// TwinCAT 3 PLC project CoreExample
// ProgramVersion: 3.1.4026.17
// libraries:
//   Tc2_Standard, * (Beckhoff Automation GmbH)
//   Tc2_System, * (Beckhoff Automation GmbH)
//   Tc3_JsonXml, * (Beckhoff Automation GmbH)
//   Tc3_Module, * (Beckhoff Automation GmbH)
//   [Twincat Open Library], * (Home)
//   VisuSymbols,3.5.10.0,System
// project tree:
//   DUTs/ ST_CameraStates.TcDUT (not stored)
//   GVLs/ Hardware_Mapping.TcGVL (not stored), Cognex_Mapping.TcGVL (not stored)
//   / PlcTask.TcTTO (not stored)
//   POUs/ MAIN.TcPOU, _5000_PRG_Aborting.TcPOU, _1000_PRG_Homing.TcPOU, _3000_PRG_Running.TcPOU, _2000_PRG_Stopping.TcPOU, _4000_PRG_Pausing.TcPOU, _6000_PRG_Proceeding.TcPOU
// real-time tasks:
//   TASK PlcTask: cycle T#10ms, priority 20, ADS port 350
//   TASK VISU_TASK: cycle T#200000us, priority 30, ADS port 351
//   TASK IO Task New: cycle T#1ms, priority 1, ADS port 301
// motion (NC):
//   TASK NC-Task 1 SAF: cycle T#2ms, priority 4, ADS port 501
//   TASK NC-Task 1 SVB: cycle T#10ms, priority 8, ADS port 511
//   AXIS Axis 1 (id 1)
//     OtherSettings: AllowMotionCmdToSlave=true
//     encoder EncType=4
//       EncPara: MaxCount=#x0000ffff
//         Inc: RefSoftSyncMask=#x0000ffff
//     drive DrvType=24
//       Analog: TorqueSetpointScale=10, ScaleFactorActTorque=0.1
//       TimeComp: TaskDelayCycles=1
//     controller CtrType=1
//       CtrPara: PriorControlFactor=1
//         Observer: BandWidth=20
//   AXIS Axis 2 (id 2)
//     OtherSettings: AllowMotionCmdToSlave=true
//     encoder EncType=4
//       EncPara: MaxCount=#x0000ffff
//         Inc: RefSoftSyncMask=#x0000ffff
//     drive DrvType=24
//       Analog: TorqueSetpointScale=10, ScaleFactorActTorque=0.1
//       TimeComp: TaskDelayCycles=1
//     controller CtrType=1
//       CtrPara: PriorControlFactor=1
//         Observer: BandWidth=20
// I/O:
//   DEVICE Device 1 (TC3 EIP Scanner), AmsNetId 172.18.236.100.2.1
//     Box 1 (In-Sight 7000 Series) // <INFO> </INFO> <EDS> C:\TwinCAT\3.1\Config\Io\EtherNetIP\02A6006401090C00.eds </EDS>
//   DEVICE Device 2 (EtherCAT), AmsNetId 172.18.236.100.3.1
//     Term 2 (EK1100) [EK1100 EtherCAT Coupler (2A E-Bus)]
//       Term 3 (EL1008) [EL1008 8Ch. Dig. Input 24V, 3ms]
//       Term 4 (EL1008) [EL1008 8Ch. Dig. Input 24V, 3ms]
//       Term 5 (EL2008) [EL2008 8Ch. Dig. Output 24V, 0.5A]
//       Term 6 (EL2008) [EL2008 8Ch. Dig. Output 24V, 0.5A]
//       Term 7 (EL7047) [EL7047 1Ch. Stepper motor output stage (50V, 5A)]
//       Term 8 (EL7047) [EL7047 1Ch. Stepper motor output stage (50V, 5A)]
//       Term 8 (EL9011) [EL9011 End Terminal]
// variable links:
//   NC-Task 1 SAF/Axes/Axis 1 <-> Device 2 (EtherCAT)/Term 2 (EK1100)/Term 7 (EL7047)
//     Drive/Inputs/In/nState1 @bit 3 <-> STM Status/Status/Error
//     Drive/Inputs/In/nState1 @bit 7 <-> STM Status/Status/Motor stall
//     Drive/Inputs/In/nState1 @bit 5 <-> STM Status/Status/Moving negative
//     Drive/Inputs/In/nState1 @bit 4 <-> STM Status/Status/Moving positive
//     Drive/Inputs/In/nState1 @bit 1 <-> STM Status/Status/Ready
//     Drive/Inputs/In/nState1 <-> STM Status/Status/Ready to enable
//     Drive/Inputs/In/nState1 @bit 6 <-> STM Status/Status/Torque reduced
//     Drive/Inputs/In/nState1 @bit 2 <-> STM Status/Status/Warning
//     Drive/Inputs/In/nState2 @bit 3 <-> STM Status/Status/Digital input 1
//     Drive/Inputs/In/nState2 @bit 4 <-> STM Status/Status/Digital input 2
//     Drive/Inputs/In/nState2 @bit 5 <-> STM Status/Status/Sync error
//     Drive/Inputs/In/nState2 @bit 7 <-> STM Status/Status/TxPDO Toggle
//     Drive/Inputs/In/nState4 @bit 1 <-> WcState/InputToggle
//     Drive/Inputs/In/nState4 <-> WcState/WcState
//     Drive/Outputs/Out/nCtrl1 <-> STM Control/Control/Enable
//     Drive/Outputs/Out/nCtrl1 @bit 2 <-> STM Control/Control/Reduce torque
//     Drive/Outputs/Out/nCtrl1 @bit 1 <-> STM Control/Control/Reset
//     Drive/Outputs/Out/nCtrl2 @bit 3 <-> STM Control/Control/Digital output 1
//     Drive/Outputs/Out/nDataOut2[0] <-> STM Velocity/Velocity
//     Enc/Inputs/In/nDataIn1[0] <-> ENC Status compact/Counter value
//     Enc/Inputs/In/nDataIn2[0] <-> ENC Status compact/Latch value
//     Enc/Inputs/In/nState1 @bit 4 <-> ENC Status compact/Status/Counter overflow
//     Enc/Inputs/In/nState1 @bit 3 <-> ENC Status compact/Status/Counter underflow
//     Enc/Inputs/In/nState1 @bit 7 <-> ENC Status compact/Status/Extrapolation stall
//     Enc/Inputs/In/nState1 <-> ENC Status compact/Status/Latch C valid
//     Enc/Inputs/In/nState1 @bit 1 <-> ENC Status compact/Status/Latch extern valid
//     Enc/Inputs/In/nState1 @bit 2 <-> ENC Status compact/Status/Set counter done
//     Enc/Inputs/In/nState2 @bit 4 <-> ENC Status compact/Status/Status of extern latch
//     Enc/Inputs/In/nState2 <-> ENC Status compact/Status/Status of input A
//     Enc/Inputs/In/nState2 @bit 1 <-> ENC Status compact/Status/Status of input B
//     Enc/Inputs/In/nState2 @bit 2 <-> ENC Status compact/Status/Status of input C
//     Enc/Inputs/In/nState2 @bit 5 <-> ENC Status compact/Status/Sync error
//     Enc/Inputs/In/nState2 @bit 7 <-> ENC Status compact/Status/TxPDO Toggle
//     Enc/Inputs/In/nState4 @bit 1 <-> WcState/InputToggle
//     Enc/Inputs/In/nState4 <-> WcState/WcState
//     Enc/Outputs/Out/nCtrl1 <-> ENC Control compact/Control/Enable latch C
//     Enc/Outputs/Out/nCtrl1 @bit 3 <-> ENC Control compact/Control/Enable latch extern on negative edge
//     Enc/Outputs/Out/nCtrl1 @bit 1 <-> ENC Control compact/Control/Enable latch extern on positive edge
//     Enc/Outputs/Out/nCtrl1 @bit 2 <-> ENC Control compact/Control/Set counter
//     Enc/Outputs/Out/nDataOut1[0] <-> ENC Control compact/Set counter value
//   NC-Task 1 SAF/Axes/Axis 2 <-> Device 2 (EtherCAT)/Term 2 (EK1100)/Term 8 (EL7047)
//     Drive/Inputs/In/nState1 @bit 3 <-> STM Status/Status/Error
//     Drive/Inputs/In/nState1 @bit 7 <-> STM Status/Status/Motor stall
//     Drive/Inputs/In/nState1 @bit 5 <-> STM Status/Status/Moving negative
//     Drive/Inputs/In/nState1 @bit 4 <-> STM Status/Status/Moving positive
//     Drive/Inputs/In/nState1 @bit 1 <-> STM Status/Status/Ready
//     Drive/Inputs/In/nState1 <-> STM Status/Status/Ready to enable
//     Drive/Inputs/In/nState1 @bit 6 <-> STM Status/Status/Torque reduced
//     Drive/Inputs/In/nState1 @bit 2 <-> STM Status/Status/Warning
//     Drive/Inputs/In/nState2 @bit 3 <-> STM Status/Status/Digital input 1
//     Drive/Inputs/In/nState2 @bit 4 <-> STM Status/Status/Digital input 2
//     Drive/Inputs/In/nState2 @bit 5 <-> STM Status/Status/Sync error
//     Drive/Inputs/In/nState2 @bit 7 <-> STM Status/Status/TxPDO Toggle
//     Drive/Inputs/In/nState4 @bit 1 <-> WcState/InputToggle
//     Drive/Inputs/In/nState4 <-> WcState/WcState
//     Drive/Outputs/Out/nCtrl1 <-> STM Control/Control/Enable
//     Drive/Outputs/Out/nCtrl1 @bit 2 <-> STM Control/Control/Reduce torque
//     Drive/Outputs/Out/nCtrl1 @bit 1 <-> STM Control/Control/Reset
//     Drive/Outputs/Out/nCtrl2 @bit 3 <-> STM Control/Control/Digital output 1
//     Drive/Outputs/Out/nDataOut2[0] <-> STM Velocity/Velocity
//     Enc/Inputs/In/nDataIn1[0] <-> ENC Status compact/Counter value
//     Enc/Inputs/In/nDataIn2[0] <-> ENC Status compact/Latch value
//     Enc/Inputs/In/nState1 @bit 4 <-> ENC Status compact/Status/Counter overflow
//     Enc/Inputs/In/nState1 @bit 3 <-> ENC Status compact/Status/Counter underflow
//     Enc/Inputs/In/nState1 @bit 7 <-> ENC Status compact/Status/Extrapolation stall
//     Enc/Inputs/In/nState1 <-> ENC Status compact/Status/Latch C valid
//     Enc/Inputs/In/nState1 @bit 1 <-> ENC Status compact/Status/Latch extern valid
//     Enc/Inputs/In/nState1 @bit 2 <-> ENC Status compact/Status/Set counter done
//     Enc/Inputs/In/nState2 @bit 4 <-> ENC Status compact/Status/Status of extern latch
//     Enc/Inputs/In/nState2 <-> ENC Status compact/Status/Status of input A
//     Enc/Inputs/In/nState2 @bit 1 <-> ENC Status compact/Status/Status of input B
//     Enc/Inputs/In/nState2 @bit 2 <-> ENC Status compact/Status/Status of input C
//     Enc/Inputs/In/nState2 @bit 5 <-> ENC Status compact/Status/Sync error
//     Enc/Inputs/In/nState2 @bit 7 <-> ENC Status compact/Status/TxPDO Toggle
//     Enc/Inputs/In/nState4 @bit 1 <-> WcState/InputToggle
//     Enc/Inputs/In/nState4 <-> WcState/WcState
//     Enc/Outputs/Out/nCtrl1 <-> ENC Control compact/Control/Enable latch C
//     Enc/Outputs/Out/nCtrl1 @bit 3 <-> ENC Control compact/Control/Enable latch extern on negative edge
//     Enc/Outputs/Out/nCtrl1 @bit 1 <-> ENC Control compact/Control/Enable latch extern on positive edge
//     Enc/Outputs/Out/nCtrl1 @bit 2 <-> ENC Control compact/Control/Set counter
//     Enc/Outputs/Out/nDataOut1[0] <-> ENC Control compact/Set counter value
//   CoreExample/CoreExample Instance <-> Device 1 (TC3 EIP Scanner)/Box 1 (In-Sight 7000 Series)
//     PlcTask Inputs/Cognex_Mapping.inpAcquiring <-> Connection 1 (Input/Output)/Inputs/Acquiring
//     PlcTask Inputs/Cognex_Mapping.inpAcquisitionID <-> Connection 1 (Input/Output)/Inputs/Acquisition ID
//     PlcTask Inputs/Cognex_Mapping.inpCommandComplete <-> Connection 1 (Input/Output)/Inputs/Command Complete
//     PlcTask Inputs/Cognex_Mapping.inpCommandExecuting <-> Connection 1 (Input/Output)/Inputs/Command Executing
//     PlcTask Inputs/Cognex_Mapping.inpCommandFailed <-> Connection 1 (Input/Output)/Inputs/Command Failed
//     PlcTask Inputs/Cognex_Mapping.inpCurrentJobID <-> Connection 1 (Input/Output)/Inputs/Current Job ID
//     PlcTask Inputs/Cognex_Mapping.inpExposureComplete <-> Connection 1 (Input/Output)/Inputs/Exposure Complete
//     PlcTask Inputs/Cognex_Mapping.inpInspecting <-> Connection 1 (Input/Output)/Inputs/Inspecting
//     PlcTask Inputs/Cognex_Mapping.inpInspectionComplete <-> Connection 1 (Input/Output)/Inputs/Inspection Complete
//     PlcTask Inputs/Cognex_Mapping.inpInspectionID <-> Connection 1 (Input/Output)/Inputs/Inspection ID
//     PlcTask Inputs/Cognex_Mapping.inpInspectionResultCode <-> Connection 1 (Input/Output)/Inputs/Inspection Result Code
//     PlcTask Inputs/Cognex_Mapping.inpInspectionResults <-> Connection 1 (Input/Output)/Inputs/Inspection Results
//     PlcTask Inputs/Cognex_Mapping.inpJobPass <-> Connection 1 (Input/Output)/Inputs/Job Pass
//     PlcTask Inputs/Cognex_Mapping.inpMissedAcq <-> Connection 1 (Input/Output)/Inputs/Missed Acq
//     PlcTask Inputs/Cognex_Mapping.inpOfflineReason <-> Connection 1 (Input/Output)/Inputs/Offline Reason
//     PlcTask Inputs/Cognex_Mapping.inpOnline <-> Connection 1 (Input/Output)/Inputs/Online
//     PlcTask Inputs/Cognex_Mapping.inpResultsBufferOverrun <-> Connection 1 (Input/Output)/Inputs/Results Buffer Overrun
//     PlcTask Inputs/Cognex_Mapping.inpResultsValid <-> Connection 1 (Input/Output)/Inputs/Results Valid
//     PlcTask Inputs/Cognex_Mapping.inpTestRunReady <-> Connection 1 (Input/Output)/Inputs/Test Run Ready
//     PlcTask Inputs/Cognex_Mapping.inpTriggerAck <-> Connection 1 (Input/Output)/Inputs/Trigger Ack
//     PlcTask Inputs/Cognex_Mapping.inpTriggerReady <-> Connection 1 (Input/Output)/Inputs/Trigger Ready
//     PlcTask Outputs/Cognex_Mapping.outBufferResultsEnable <-> Connection 1 (Input/Output)/Outputs/Buffer Results Enable
//     PlcTask Outputs/Cognex_Mapping.outCommand <-> Connection 1 (Input/Output)/Outputs/Command
//     PlcTask Outputs/Cognex_Mapping.outExecuteCommand <-> Connection 1 (Input/Output)/Outputs/Execute Command
//     PlcTask Outputs/Cognex_Mapping.outInspectionResultsAck <-> Connection 1 (Input/Output)/Outputs/Inspection Results Ack
//     PlcTask Outputs/Cognex_Mapping.outSetOffline <-> Connection 1 (Input/Output)/Outputs/Set Offline
//     PlcTask Outputs/Cognex_Mapping.outSoftEvent{0..7} <-> Connection 1 (Input/Output)/Outputs/Soft Event {0..7}  (8 links)
//     PlcTask Outputs/Cognex_Mapping.outTriggerCamera <-> Connection 1 (Input/Output)/Outputs/Trigger
//     PlcTask Outputs/Cognex_Mapping.outTriggerEnable <-> Connection 1 (Input/Output)/Outputs/Trigger Enable
//     PlcTask Outputs/Cognex_Mapping.outUserData <-> Connection 1 (Input/Output)/Outputs/User Data
//   CoreExample/CoreExample Instance <-> Device 2 (EtherCAT)/Term 2 (EK1100)/Term 3 (EL1008)
//     PlcTask Inputs/Cognex_Mapping.input1 <-> Channel 1/Input
//     PlcTask Inputs/Cognex_Mapping.input2 <-> Channel 2/Input
//   CoreExample/CoreExample Instance <-> Device 2 (EtherCAT)/Term 2 (EK1100)/Term 5 (EL2008)
//     PlcTask Outputs/Cognex_Mapping.output1 <-> Channel 1/Output
//     PlcTask Outputs/Cognex_Mapping.output2 <-> Channel 2/Output

// ---- POUs/MAIN.TcPOU
PROGRAM MAIN
VAR
    fbStateMachine : FB_StateMachine;
    
    // Online-view command buttons — set TRUE in watch/online to trigger, auto-reset each scan
    btnHome    : BOOL;
    btnStart   : BOOL;
    btnStop    : BOOL;
    btnAbort   : BOOL;
    btnPause   : BOOL;
    btnProceed : BOOL;
    btnRetry   : BOOL;
END_VAR

fbStateMachine(
    EnableIn := TRUE,
    cfgAutoRun := FALSE  // disable auto-run so manual buttons stay in control
);

// --- Online command buttons (write TRUE in TwinCAT online view to trigger) ---
IF btnHome    THEN fbStateMachine.Home();    btnHome    := FALSE; END_IF;
IF btnStart   THEN fbStateMachine.Start();   btnStart   := FALSE; END_IF;
IF btnStop    THEN fbStateMachine.Stop();    btnStop    := FALSE; END_IF;
IF btnAbort   THEN fbStateMachine.Abort();   btnAbort   := FALSE; END_IF;
IF btnPause   THEN fbStateMachine.Pause();   btnPause   := FALSE; END_IF;
IF btnProceed THEN fbStateMachine.Proceed(); btnProceed := FALSE; END_IF;
IF btnRetry   THEN fbStateMachine.Retry();   btnRetry   := FALSE; END_IF;

_1000_PRG_Homing(sm := fbStateMachine);
_3000_PRG_Running(sm := fbStateMachine);
_2000_PRG_Stopping(sm := fbStateMachine);
_5000_PRG_Aborting(sm := fbStateMachine);
_4000_PRG_Pausing(sm := fbStateMachine);
_6000_PRG_Proceeding(sm := fbStateMachine);

END_PROGRAM

// ---- POUs/_1000_PRG_Homing.TcPOU
PROGRAM _1000_PRG_Homing
VAR_IN_OUT
    sm : FB_StateMachine;
END_VAR
VAR
    step1000 : FB_Step;
    step1002 : FB_Step;
    step1004 : FB_Step;

    // Simulated hardware signals
    bDriveEnabled      : BOOL;
    bHomeSensorReached : BOOL;
    bServoReady        : BOOL;
    nRetryCount        : INT;
    tonHomeDelay       : TON;
END_VAR


//=============================================================================
// STEP 1000 - Initialize Homing
// Demonstrates: Entry (one-shot initialization), Execute (wait for perms),
//               Exiting (cleanup before advancing)
//=============================================================================
step1000(sm := sm, nStep := 1000, nNextStep := 1002, nTimeout := 10, sName := 'Init Homing');

IF step1000.Entry THEN
    // One-shot: reset state from any prior attempt
    bDriveEnabled := FALSE;
    bHomeSensorReached := FALSE;
    nRetryCount := 0;
    tonHomeDelay(IN := FALSE);  // reset timer
END_IF;

IF step1000.Execute THEN
    // Simulate: enable drive after a short delay
    tonHomeDelay(IN := TRUE, PT := T#2S);
    bDriveEnabled := tonHomeDelay.Q;

    // Permissives gate the transition to next step
    step1000.MapPerm(nIndex := 0, sDescription := 'Drive Enabled',      bValue := bDriveEnabled);
    step1000.MapPerm(nIndex := 1, sDescription := 'Safety Circuit OK',  bValue := TRUE);
    step1000.MapPerm(nIndex := 2, sDescription := 'No Active Faults',   bValue := TRUE);
END_IF;

IF step1000.Exiting THEN
    // One-shot cleanup: latch that initialization is done
    tonHomeDelay(IN := FALSE);
END_IF;

//=============================================================================
// STEP 1002 - Execute Homing Move
// Demonstrates: Entry (command actuator), Execute (monitor completion),
//               SetNextStep (dynamic branching on success/failure)
//=============================================================================
step1002(sm := sm, nStep := 1002, nNextStep := 1004, nTimeout := 20, sName := 'Execute Home Move');

IF step1002.Entry THEN
    // One-shot: command the axis to home
    bHomeSensorReached := FALSE;
    bServoReady := FALSE;
END_IF;

IF step1002.Execute THEN
    // Simulate homing motion completing after some time
    bHomeSensorReached := sm.StepInfo.StepTimerSeconds >= 5.0;
    bServoReady := bHomeSensorReached;

    step1002.MapPerm(nIndex := 0, sDescription := 'Home Sensor Reached', bValue := bHomeSensorReached);
    step1002.MapPerm(nIndex := 1, sDescription := 'Servo Settled',       bValue := bServoReady);
END_IF;

IF step1002.Exiting THEN
    // Could log completion or capture final position here
    ;
END_IF;

//=============================================================================
// STEP 1004 - Verify Home Position
// Demonstrates: Simple verification step, nNextStep := 0 ends the sequence
//=============================================================================
step1004(sm := sm, nStep := 1004, nNextStep := 0, nTimeout := 5, sName := 'Verify Home Position');

IF step1004.Entry THEN
    // Nothing special to initialize
    ;
END_IF;

IF step1004.Execute THEN
    // Verify the home position is stable
    step1004.MapPerm(nIndex := 0, sDescription := 'Position Stable', bValue := sm.StepInfo.StepTimerSeconds >= 1.0);
    step1004.MapPerm(nIndex := 1, sDescription := 'Encoder Valid',   bValue := TRUE);
END_IF;

END_PROGRAM

// ---- POUs/_3000_PRG_Running.TcPOU
PROGRAM _3000_PRG_Running
VAR_IN_OUT
    sm : FB_StateMachine;
END_VAR
VAR
    step3000 : FB_Step;
    step3002 : FB_Step;
    step3004 : FB_Step;
    step3006 : FB_Step;
    step3008 : FB_Step;

    // Simulated process signals
    bMaterialLoaded    : BOOL;
    bProcessRunning    : BOOL;
    bQualityOK         : BOOL;
    bPackagingReady    : BOOL;
    nPartCount         : INT;
    nBatchTarget       : INT := 10;
    tonProcess         : TON;
    tonInspect         : TON;
END_VAR


//=============================================================================
// STEP 3000 - Load Raw Material
// Demonstrates: Entry (command loader), Execute (wait for material sensor)
//=============================================================================
step3000(sm := sm, nStep := 3000, nNextStep := 3002, nTimeout := 12, sName := 'Load Material');

IF step3000.Entry THEN
    // One-shot: command the loader to feed material
    bMaterialLoaded := FALSE;
    nPartCount := 0;
    tonProcess(IN := FALSE);
END_IF;

IF step3000.Execute THEN
    // Simulate material arriving after 3s
    bMaterialLoaded := sm.Status.Step.TimerSeconds >= 3.0;

    step3000.MapPerm(nIndex := 0, sDescription := 'Material Loaded',    bValue := bMaterialLoaded);
    step3000.MapPerm(nIndex := 1, sDescription := 'Temperature In Range', bValue := TRUE);
    step3000.MapPerm(nIndex := 2, sDescription := 'Recipe Selected',    bValue := TRUE);
END_IF;

IF step3000.Exiting THEN
    // Material confirmed, clear loader command
    ;
END_IF;

//=============================================================================
// STEP 3002 - Run Production Cycle
// Demonstrates: Entry (start process), Execute (count parts), Exiting (stop)
//=============================================================================
step3002(sm := sm, nStep := 3002, nNextStep := 3004, nTimeout := 30, sName := 'Run Cycle');

IF step3002.Entry THEN
    bProcessRunning := FALSE;
    tonProcess(IN := FALSE);
END_IF;

IF step3002.Execute THEN
    // Simulate process running, completes after 5s
    tonProcess(IN := TRUE, PT := T#5S);
    bProcessRunning := TRUE;
    nPartCount := nPartCount + 1;  // In real code this would be edge-triggered

    step3002.MapPerm(nIndex := 0, sDescription := 'Cycle Complete',   bValue := tonProcess.Q);
    step3002.MapPerm(nIndex := 1, sDescription := 'No Alarms Active', bValue := TRUE);
END_IF;

IF step3002.Exiting THEN
    tonProcess(IN := FALSE);
    bProcessRunning := FALSE;
END_IF;

//=============================================================================
// STEP 3004 - Quality Inspection
// Demonstrates: Inline dynamic branching via nNextStep (pass -> pack, fail -> finalize).
// nNextStep is re-evaluated every scan, so a SEL / IF computed before the call
// is all you need -- no override method, no init-time registration.
//=============================================================================
step3004(sm := sm,
         nStep     := 3004,
         nNextStep := SEL(bQualityOK, 3008, 3006),   // fail -> skip packaging
         nTimeout  := 12,
         sName     := 'Quality Inspection');

IF step3004.Entry THEN
    bQualityOK := FALSE;
    tonInspect(IN := FALSE);
END_IF;

IF step3004.Execute THEN
    // Simulate inspection taking 2s, always passes in this example
    tonInspect(IN := TRUE, PT := T#2S);
    bQualityOK := tonInspect.Q;

    step3004.MapPerm(nIndex := 0, sDescription := 'Inspection Complete', bValue := tonInspect.Q);
END_IF;

IF step3004.Exiting THEN
    tonInspect(IN := FALSE);
END_IF;

//=============================================================================
// STEP 3006 - Package Product
// Demonstrates: Entry (prepare packaging), Execute (seal & label)
//=============================================================================
step3006(sm := sm, nStep := 3006, nNextStep := 3008, nTimeout := 15, sName := 'Package Product');

IF step3006.Entry THEN
    bPackagingReady := FALSE;
END_IF;

IF step3006.Execute THEN
    bPackagingReady := sm.Status.Step.TimerSeconds >= 3.0;

    step3006.MapPerm(nIndex := 0, sDescription := 'Box Sealed',   bValue := bPackagingReady);
    step3006.MapPerm(nIndex := 1, sDescription := 'Label Applied', bValue := bPackagingReady);
    step3006.MapPerm(nIndex := 2, sDescription := 'Conveyor Clear', bValue := TRUE);
END_IF;

IF step3006.Exiting THEN
    // Package dispatched
    ;
END_IF;

//=============================================================================
// STEP 3008 - Finalize Batch
// Demonstrates: Exiting (generate reports), nNextStep := 0 ends sequence
//=============================================================================
step3008(sm := sm, nStep := 3008, nNextStep := 0, nTimeout := 10, sName := 'Finalize Batch');

IF step3008.Execute THEN
    step3008.MapPerm(nIndex := 0, sDescription := 'Batch Record Saved', bValue := sm.Status.Step.TimerSeconds >= 2.0);
    step3008.MapPerm(nIndex := 1, sDescription := 'Counters Reset',     bValue := TRUE);
END_IF;

IF step3008.Exiting THEN
    // Final cleanup: reset batch counters
    nPartCount := 0;
END_IF;

END_PROGRAM

// ---- POUs/_2000_PRG_Stopping.TcPOU
PROGRAM _2000_PRG_Stopping
VAR_IN_OUT
    sm : FB_StateMachine;
END_VAR
VAR
    step2000 : FB_Step;
    step2002 : FB_Step;
    step2004 : FB_Step;

    // Simulated signals
    bMotorsStopped     : BOOL;
    bConveyorEmpty     : BOOL;
    bBrakeEngaged      : BOOL;
    tonDecel           : TON;
END_VAR


//=============================================================================
// STEP 2000 - Controlled Deceleration
// Demonstrates: Entry (command stop), Execute (monitor decel), Exiting (confirm)
//=============================================================================
step2000(sm := sm, nStep := 2000, nNextStep := 2002, nTimeout := 10, sName := 'Decelerate');

IF step2000.Entry THEN
    // One-shot: command all axes to decelerate
    bMotorsStopped := FALSE;
    bBrakeEngaged := FALSE;
    tonDecel(IN := FALSE);
END_IF;

IF step2000.Execute THEN
    // Simulate controlled deceleration over 4 seconds
    tonDecel(IN := TRUE, PT := T#4S);
    bMotorsStopped := tonDecel.Q;

    step2000.MapPerm(nIndex := 0, sDescription := 'Motors Stopped',   bValue := bMotorsStopped);
    step2000.MapPerm(nIndex := 1, sDescription := 'No Motion Faults', bValue := TRUE);
END_IF;

IF step2000.Exiting THEN
    tonDecel(IN := FALSE);
END_IF;

//=============================================================================
// STEP 2002 - Clear Conveyor
// Demonstrates: Entry (start flush), Execute (wait empty), Exiting (disengage)
//=============================================================================
step2002(sm := sm, nStep := 2002, nNextStep := 2004, nTimeout := 15, sName := 'Clear Conveyor');

IF step2002.Entry THEN
    bConveyorEmpty := FALSE;
END_IF;

IF step2002.Execute THEN
    // Simulate conveyor clearing in 6 seconds
    bConveyorEmpty := sm.StepInfo.StepTimerSeconds >= 6.0;

    step2002.MapPerm(nIndex := 0, sDescription := 'Conveyor Empty',      bValue := bConveyorEmpty);
    step2002.MapPerm(nIndex := 1, sDescription := 'Product Accounted For', bValue := TRUE);
END_IF;

IF step2002.Exiting THEN
    // Conveyor off
    ;
END_IF;

//=============================================================================
// STEP 2004 - Engage Brakes & Safe State
// Demonstrates: Entry (engage brakes), nNextStep := 0 completes sequence
//=============================================================================
step2004(sm := sm, nStep := 2004, nNextStep := 0, nTimeout := 5, sName := 'Engage Brakes');

IF step2004.Entry THEN
    bBrakeEngaged := FALSE;
END_IF;

IF step2004.Execute THEN
    bBrakeEngaged := sm.StepInfo.StepTimerSeconds >= 1.0;

    step2004.MapPerm(nIndex := 0, sDescription := 'Brakes Engaged',   bValue := bBrakeEngaged);
    step2004.MapPerm(nIndex := 1, sDescription := 'Safe State Active', bValue := TRUE);
END_IF;

END_PROGRAM

// ---- POUs/_5000_PRG_Aborting.TcPOU
PROGRAM _5000_PRG_Aborting
VAR_IN_OUT
    sm : FB_StateMachine;
END_VAR
VAR
    step5000 : FB_Step;
    step5002 : FB_Step;
    step5004 : FB_Step;

    // Emergency signals
    bOutputsDisabled   : BOOL;
    bPneumaticsVented  : BOOL;
    bMotionHalted      : BOOL;
    tonEmergency       : TON;
END_VAR


//=============================================================================
// STEP 5000 - Immediate Halt
// Demonstrates: Entry (kill outputs immediately), Execute (verify halted)
// NOTE: Abort is an emergency path — minimal delays, prioritize safety
//=============================================================================
step5000(sm := sm, nStep := 5000, nNextStep := 5002, nTimeout := 3, sName := 'Immediate Halt');

IF step5000.Entry THEN
    // One-shot: immediately disable all outputs
    bOutputsDisabled := TRUE;   // In real code: write FALSE to all DO
    bMotionHalted := FALSE;
    tonEmergency(IN := FALSE);
END_IF;

IF step5000.Execute THEN
    // Verify motion has actually stopped (simulate 1s settling)
    tonEmergency(IN := TRUE, PT := T#1S);
    bMotionHalted := tonEmergency.Q;

    step5000.MapPerm(nIndex := 0, sDescription := 'Outputs Disabled', bValue := bOutputsDisabled);
    step5000.MapPerm(nIndex := 1, sDescription := 'Motion Halted',    bValue := bMotionHalted);
END_IF;

IF step5000.Exiting THEN
    tonEmergency(IN := FALSE);
END_IF;

//=============================================================================
// STEP 5002 - Vent Pneumatics
// Demonstrates: Entry (open vent valves), Execute (wait for pressure drop)
//=============================================================================
step5002(sm := sm, nStep := 5002, nNextStep := 5004, nTimeout := 8, sName := 'Vent Pneumatics');

IF step5002.Entry THEN
    // One-shot: open all vent valves
    bPneumaticsVented := FALSE;
END_IF;

IF step5002.Execute THEN
    // Simulate pressure bleed-off over 3s
    bPneumaticsVented := sm.StepInfo.StepTimerSeconds >= 3.0;

    step5002.MapPerm(nIndex := 0, sDescription := 'Pressure Below 0.5 bar', bValue := bPneumaticsVented);
    step5002.MapPerm(nIndex := 1, sDescription := 'Vent Valves Open',       bValue := TRUE);
END_IF;

//=============================================================================
// STEP 5004 - Confirm Safe State
// Demonstrates: Exiting (log abort reason), nNextStep := 0 enters Aborted
//=============================================================================
step5004(sm := sm, nStep := 5004, nNextStep := 0, nTimeout := 5, sName := 'Confirm Safe State');

IF step5004.Execute THEN
    step5004.MapPerm(nIndex := 0, sDescription := 'All Energy Isolated',  bValue := sm.StepInfo.StepTimerSeconds >= 1.0);
    step5004.MapPerm(nIndex := 1, sDescription := 'Safety Relay Latched', bValue := TRUE);
END_IF;

IF step5004.Exiting THEN
    // Log abort event for maintenance review
    ;
END_IF;

END_PROGRAM

// ---- POUs/_4000_PRG_Pausing.TcPOU
PROGRAM _4000_PRG_Pausing
VAR_IN_OUT
    sm : FB_StateMachine;
END_VAR
VAR
    step4000 : FB_Step;
    step4002 : FB_Step;

    // Simulated signals
    bAxesHolding       : BOOL;
    bProcessSuspended  : BOOL;
    tonRampDown        : TON;
END_VAR


//=============================================================================
// STEP 4000 - Ramp Down to Hold
// Demonstrates: Entry (command hold), Execute (monitor ramp), Exiting (confirm)
//=============================================================================
step4000(sm := sm, nStep := 4000, nNextStep := 4002, nTimeout := 8, sName := 'Ramp Down');

IF step4000.Entry THEN
    // One-shot: command controlled ramp-down
    bAxesHolding := FALSE;
    bProcessSuspended := FALSE;
    tonRampDown(IN := FALSE);
END_IF;

IF step4000.Execute THEN
    // Simulate ramp-down over 3 seconds
    tonRampDown(IN := TRUE, PT := T#3S);
    bAxesHolding := tonRampDown.Q;

    step4000.MapPerm(nIndex := 0, sDescription := 'Axes Holding Position', bValue := bAxesHolding);
    step4000.MapPerm(nIndex := 1, sDescription := 'No Motion Commands',    bValue := TRUE);
END_IF;

IF step4000.Exiting THEN
    tonRampDown(IN := FALSE);
END_IF;

//=============================================================================
// STEP 4002 - Suspend Process
// Demonstrates: Entry (freeze process state), nNextStep := 0 enters Paused
//=============================================================================
step4002(sm := sm, nStep := 4002, nNextStep := 0, nTimeout := 5, sName := 'Suspend Process');

IF step4002.Entry THEN
    bProcessSuspended := FALSE;
END_IF;

IF step4002.Execute THEN
    // Simulate process freeze
    bProcessSuspended := sm.StepInfo.StepTimerSeconds >= 1.0;

    step4002.MapPerm(nIndex := 0, sDescription := 'Process State Saved',  bValue := bProcessSuspended);
    step4002.MapPerm(nIndex := 1, sDescription := 'Heaters in Standby',   bValue := TRUE);
    step4002.MapPerm(nIndex := 2, sDescription := 'Vacuum Maintained',    bValue := TRUE);
END_IF;

IF step4002.Exiting THEN
    // Process is now paused - operator can inspect / Proceed resumes
    ;
END_IF;

END_PROGRAM

// ---- POUs/_6000_PRG_Proceeding.TcPOU
PROGRAM _6000_PRG_Proceeding
VAR_IN_OUT
    sm : FB_StateMachine;
END_VAR
VAR
    step6000 : FB_Step;
    step6002 : FB_Step;
    step6004 : FB_Step;

    // Resume signals
    bHeatersReady      : BOOL;
    bMotionResynced    : BOOL;
    bProductionResumed : BOOL;
    tonWarmup          : TON;
    tonResync          : TON;
END_VAR


//=============================================================================
// STEP 6000 - Restore Process Conditions
// Demonstrates: Entry (re-enable heaters), Execute (wait for temp), Exiting
// This runs after operator presses Proceed from Paused state
//=============================================================================
step6000(sm := sm, nStep := 6000, nNextStep := 6002, nTimeout := 15, sName := 'Restore Conditions');

IF step6000.Entry THEN
    // One-shot: re-enable heaters and process systems
    bHeatersReady := FALSE;
    tonWarmup(IN := FALSE);
END_IF;

IF step6000.Execute THEN
    // Simulate heaters reaching setpoint after 4s
    tonWarmup(IN := TRUE, PT := T#4S);
    bHeatersReady := tonWarmup.Q;

    step6000.MapPerm(nIndex := 0, sDescription := 'Heaters At Setpoint', bValue := bHeatersReady);
    step6000.MapPerm(nIndex := 1, sDescription := 'Coolant Flowing',     bValue := TRUE);
    step6000.MapPerm(nIndex := 2, sDescription := 'Interlocks Satisfied', bValue := TRUE);
END_IF;

IF step6000.Exiting THEN
    tonWarmup(IN := FALSE);
END_IF;

//=============================================================================
// STEP 6002 - Re-synchronize Motion
// Demonstrates: Entry (command resync), Execute (verify position match)
//=============================================================================
step6002(sm := sm, nStep := 6002, nNextStep := 6004, nTimeout := 10, sName := 'Resync Motion');

IF step6002.Entry THEN
    bMotionResynced := FALSE;
    tonResync(IN := FALSE);
END_IF;

IF step6002.Execute THEN
    // Simulate motion resync over 2s
    tonResync(IN := TRUE, PT := T#2S);
    bMotionResynced := tonResync.Q;

    step6002.MapPerm(nIndex := 0, sDescription := 'Axes Synchronized', bValue := bMotionResynced);
    step6002.MapPerm(nIndex := 1, sDescription := 'Position Error OK', bValue := TRUE);
END_IF;

IF step6002.Exiting THEN
    tonResync(IN := FALSE);
END_IF;

//=============================================================================
// STEP 6004 - Resume Production
// Demonstrates: Entry (restart process), Exiting (hand back to Running)
//=============================================================================
step6004(sm := sm, nStep := 6004, nNextStep := 0, nTimeout := 5, sName := 'Resume Production');

IF step6004.Entry THEN
    bProductionResumed := FALSE;
END_IF;

IF step6004.Execute THEN
    bProductionResumed := sm.StepInfo.StepTimerSeconds >= 1.0;

    step6004.MapPerm(nIndex := 0, sDescription := 'Process Restarted',  bValue := bProductionResumed);
    step6004.MapPerm(nIndex := 1, sDescription := 'Output Rate Normal', bValue := TRUE);
END_IF;

IF step6004.Exiting THEN
    // Handoff complete - SM transitions back to Running
    ;
END_IF;

END_PROGRAM
